(*These are axis parameters that are set up during commissioning and
in theory don't neeed to be change as part of daily moving of axes.
For instance they may be changed due to poor parameter selection
or change of instrument configuration.*)
TYPE ST_AxisConfig_1 :
STRUCT
    //Axis Parameters
    fOverride: LREAL := 100; //Controller override %, used a global scale for an axis in terms of velocity. Generally set to 100%.
    fHomePosition: LREAL := 0; //The position that the axis should be set to once homing is completed
    fHomeFinishDistance: LREAL := 0; //Distrance that the axis should move back into the working zone after homing is finished
    eHomeSeq: E_HomingRoutines; //Homing sequence to perform
    eRestorePosition: E_RestorePosition; //Restore position of incremental axis after loss of power to the CPU, 0=don't restore, 1=restore but don't home

    //Read and Write parameters
    eAxisParameters: E_AxisParameters; //Enumeration of axis parameters
    fWriteAxisParameter: LREAL; //The value to be writen to eAxisParameterNumber
    fReadAxisParameter: LREAL; //Read the current value of the selected eAxisParameterNumber
    bReadAxisParameterValid: BOOL; //Is the current data thats been read valid value

    //Single master axis parameters
    stMasterAxis: ST_GearAxis; //A reference to the axis that this is a slave of
    afSlaveAxisRatio: ARRAY [1..GVL_APP.nAXIS_NUM] OF LREAL; //The gearing between this axis as a master and any slaves. e.g. if this is a 1 to 1 master of axis 2 this will be [0, 1, 0 ...]

    //Multi master axis parameters
    astMultiMasterAxis: ARRAY [1..4] OF ST_GearAxis;
    astMultiMasterAxisLatched: ARRAY [1..4] OF ST_GearAxis; //A kind of readback since one doesn't exist in AXIS_REF
    afMultiSlaveAxisRatio: ARRAY [1..GVL_APP.nAXIS_NUM] OF LREAL;

    // Read only MC parameters
    bReadMcParametersValid: BOOL:= FALSE;
    bReadMcParametersError: BOOL:= FALSE;
    fVelocityDefaultSlow: LREAL; //Read only - AxisVeloManSlow
    fVelocityDefaultFast: LREAL; //Read only - AxisVeloManFast
    fHomingVelToCam: LREAL; //Read only - AxisCalibrationVelocityForward
    fHomingVelFromCam: LREAL; //Read only - AxisCalibrationVelocityBackward
    fVeloMax: LREAL; //Read only - fVeloMax
    fDefaultAcc: LREAL; //Read only - AxisAcc
    fDefaultDec: LREAL; //Read only - AxisDec
    bEnMinSoftPosLimit: BOOL; //Read only
    fMinSoftPosLimit: LREAL; //Read only
    bEnMaxSoftPosLimit: BOOL; //Read only
    fMaxSoftPosLimit: LREAL; //Read only
    bEnPositionLagMonitoring: BOOL; //Read only
    fMaxPosLagValue: LREAL; //Read only
    bEnTargetPositionMonitoring: BOOL; //Read only
    fTargetPositionWindow: LREAL; //Read only
END_STRUCT
END_TYPE

(* stored: Version 1.1.0.1, ProductVersion 3.1.4024.6
   DUT ST_AxisConfig_1: Id {c1627b51-a843-453c-9ab0-b0e6aaa840dd} *)
